FUNCTION_BLOCK E_SELECT
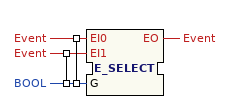
  EVENT_INPUT
    EI0 WITH G;
    EI1 WITH G;
  END_EVENT
  EVENT_OUTPUT
    EO;
  END_EVENT
  VAR_INPUT
    G : BOOL;
  END_VAR
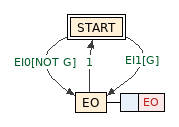
  EC_STATES
    START;
    EO : -> EO;
  END_STATES
  EC_TRANSITIONS
    EO TO START := 1;
    START TO EO := EI0[NOT G];
    START TO EO := EI1[G];
  END_TRANSITIONS
END_FUNCTION_BLOCK
